(* Logix 5000 project; controller GP1 vendor 1 type 14 code 155 rev 32.11; software revision 32.01 *)
// GP1

TASK MainTask (continuous, watchdog 500 ms) : MainProgram

MODULES
   Local : vendor 1 type 14 code 155 (PointIO 0, rev 32.11)
      GP1_INPUT_MODULE_4 : 1734-IB8 (PointIO 4, rev 3.1, Input RPI 20 ms)
           Local:4:I.Data.1   // IC TOPE
           Local:4:I.Data.0   // FC TOPE
           Local:4:I.Data.3   // CAPACITIVO IZQUIERDO
           Local:4:I.Data.6   // CAPACITIVO DERECHO
      GP1_INPUT_MODULE_5 : 1734-IB8 (PointIO 5, rev 3.1, Input RPI 20 ms)
           Local:5:I.Data.2   // ARRANQUE
           Local:5:I.Data.3   // BOTON REARME
           Local:5:I.Data.1   // PARO
           Local:5:I.Data.0   // INDUCTIVO TOPE
      Discrete_IO : Embedded (PointIO 1, rev 32.11, Output RPI 20 ms)
           Local:1:I.Data.5   // IC CLAMP HORIZONTAL
           Local:1:I.Data.7   // IC CLAMP VERTICAL
           Local:1:I.Data.8   // IC NAVAJAS 3 R
           Local:1:I.Data.10   // IC CLAMP
           Local:1:I.Data.11   // FC CLAMP
           Local:1:I.Data.9   // FC NAVAJAS 3 R
           Local:1:I.Data.6   // FC CLAMP VERTICAL
           Local:1:I.Data.0   // FC NAVAJA 1
           Local:1:I.Data.1   // IC NAVAJA 1
           Local:1:I.Data.15   // FC TROQUEL
           Local:1:I.Data.2   // IC NAVAJAS 3 L
           Local:1:I.Data.4   // FC CLAMP HORIZONTAL
           Local:1:I.Data.3   // FC NAVAJAS 3 L
           Local:1:I.Data.14   // IC TROQUEL
           Local:1:I.Data.12   // FC CORTE SUPERIOR
           Local:1:I.Data.13   // IC CORTE SUPERIOR
           Local:1:O.Data.15   // GREEN
      GP1_OUTPUT_MODULE_3 : 1734-OB8 (PointIO 3, rev 3.1, Output RPI 20 ms)
      GP1_OUTPUT_MODULE_2 : 1734-OB8 (PointIO 2, rev 3.1, Output RPI 20 ms)
           Local:2:O.Data.0   // YELLOW
           Local:2:O.Data.1   // RED
           Local:2:O.Data.2   // AZUL
END_MODULES

VAR_GLOBAL   (* controller tags *)
   ACT0_OFF : BOOL := 1;   // NAVAJAS 3 R OFF
   ACT0_ON : BOOL;   // NAVAJAS 3 R ON
   ACT1_OFF : BOOL := 1;   // TROQUEL OFF
   ACT1_ON : BOOL;   // TROQUEL ON
   ACT2_OFF : BOOL := 1;   // CORTE SUPERIOR OFF
   ACT2_ON : BOOL;   // CORTE SUPERIOR ON
   ACT3_OFF : BOOL := 1;   // NAVAJA 1 OFF
   ACT3_ON : BOOL;   // NAVAJA 1 ON
   ACT4_OFF : BOOL;   // CLAMP VERTICAL OFF
   ACT4_ON : BOOL;   // CLAMP VERTICAL ON
   ACT5_OFF : BOOL := 1;   // CLAMP OFF
   ACT5_ON : BOOL;   // CLAMP ON
   ACT6_OFF : BOOL;   // CLAMP HORIZONTAL OFF
   ACT6_ON : BOOL;   // CLAMP HORIZONTAL ON
   ACT7_OFF : BOOL := 1;   // NAVAJA 3 L OFF
   ACT7_ON : BOOL;   // NAVAJA 3 L ON
   ACT8_OFF : BOOL;   // TOPE OFF
   ACT8_ON : BOOL := 1;   // TOPE ON
   AIR_ALARM : BOOL;
   ALARM_TIM : TIMER := (PRE := 5000);
   ALARMED : BOOL := 1;
   ARRANQUE_AUTO : BOOL;
   AUTO : BOOL;
   C1 : COUNTER := (ACC := 14, CU := 1, DN := 1);
   CAPACITIVE_SENSOR_1 : BOOL;
   CAPACITIVE_SENSOR_2 : BOOL;
   CND1 : BOOL;
   CND10 : BOOL;
   CND2 : BOOL;
   CND3 : BOOL;
   CND4 : BOOL;
   CND5 : BOOL;
   CND6 : BOOL;
   CND7 : BOOL;
   CND8 : BOOL;
   CND9 : BOOL;
   CORTE_VALVULA : BOOL := 1;
   CORTINA_SEG : BOOL;
   CT : COUNTER := (ACC := 9999);
   CURRENT_SCREEN : DINT;
   E_STOP : BOOL := 1;
   E_STOP_ALARM : BOOL := 1;
   EstadoHMI : DINT := 3;
   EVBI0_AUTO_OFF : BOOL;   // NAVAJAS 3 OFF AUTO
   EVBI0_AUTO_ON : BOOL;   // NAVAJAS 3 ON AUTO
   EVBI0_MAN_OFF : BOOL;   // NAVAJAS 3 OFF MANUAL
   EVBI0_MAN_ON : BOOL;   // NAVAJAS 3 ON MANUAL
   EVBI0_OFF : BOOL;   // NAVAJAS 3 OFF
   EVBI0_ON : BOOL;   // NAVAJAS 3 ON
   EVBI1_AUTO_OFF : BOOL;   // TROQUEL OFF AUTO
   EVBI1_AUTO_ON : BOOL;   // TROQUEL ON AUTO
   EVBI1_MAN_OFF : BOOL;   // TROQUEL OFF MANUAL
   EVBI1_MAN_ON : BOOL;   // TROQUEL ON MANUAL
   EVBI1_OFF : BOOL;   // TROQUEL OFF
   EVBI1_ON : BOOL;   // TROQUEL ON
   EVBI2_AUTO_OFF : BOOL;   // CLAMP OFF AUTO
   EVBI2_AUTO_ON : BOOL;   // CLAMP ON AUTO
   EVBI2_MAN_OFF : BOOL;   // CLAMP OFF MANUAL
   EVBI2_MAN_ON : BOOL;   // CLAMP ON MANUAL
   EVBI2_OFF : BOOL;   // CLAMP OFF
   EVBI2_ON : BOOL;   // CLAMP ON
   EVBI3_AUTO_OFF : BOOL;   // NAVAJA 1 OFF AUTO
   EVBI3_AUTO_ON : BOOL;   // NAVAJA 1 ON AUTO
   EVBI3_MAN_OFF : BOOL;   // NAVAJA 1 OFF MANUAL
   EVBI3_MAN_ON : BOOL;   // NAVAJA 1 ON MANUAL
   EVBI3_OFF : BOOL;   // NAVAJA 1 OFF
   EVBI3_ON : BOOL;   // NAVAJA 1 ON
   EVBI4_AUTO_OFF : BOOL;   // CLAMP VERTICAL OFF AUTO
   EVBI4_AUTO_ON : BOOL;   // CLAMP VERTICAL ON AUTO
   EVBI4_MAN_OFF : BOOL;   // CLAMP VERTICAL OFF MANUAL
   EVBI4_MAN_ON : BOOL;   // CLAMP VERTICAL ON MANUAL
   EVBI4_OFF : BOOL;   // CLAMP VERTICAL OFF
   EVBI4_ON : BOOL;   // CLAMP VERTICAL ON
   EVBI5_AUTO_OFF : BOOL;   // CORTE SUPERIOR OFF AUTO
   EVBI5_AUTO_ON : BOOL;   // CORTE SUPERIOR ON AUTO
   EVBI5_MAN_OFF : BOOL;   // CORTE SUPERIOR OFF MANUAL
   EVBI5_MAN_ON : BOOL;   // CORTE SUPERIOR ON MANUAL
   EVBI5_OFF : BOOL;   // CORTE SUPERIOR OFF
   EVBI5_ON : BOOL;   // CORTE SUPERIOR ON
   EVBI6_AUTO_OFF : BOOL;   // CLAMP HORIZONTAL OFF AUTO
   EVBI6_AUTO_ON : BOOL;   // CLAMP HORIZONTAL ON AUTO
   EVBI6_MAN_OFF : BOOL;   // CLAMP HORIZONTAL OFF MANUAL
   EVBI6_MAN_ON : BOOL;   // CLAMP HORIZONTAL ON MANUAL
   EVBI6_OFF : BOOL;   // CLAMP HORIZONTAL OFF
   EVBI6_ON : BOOL;   // CLAMP HORIZONTAL ON
   EVMONO1_AUTO_OFF : BOOL;
   EVMONO1_AUTO_ON : BOOL;   // TOPE_AUTO_ON
   EVMONO1_MAN_OFF : BOOL;
   EVMONO1_MAN_ON : BOOL;
   EVMONO_OFF : BOOL;
   EVMONO_ON : BOOL;   // TOPE ON
   EXCEDDED_TIME_FOR_CILINDERS : BOOL;
   EXCEDDED_TIME_FOR_INIT_COND : BOOL;
   FAIL_COUNT : COUNTER;
   GREEN_LIGHT : BOOL;
   INITIAL_CONDITIONS_NOT_READY : BOOL := 1;
   INITIAL_CONDITIONS_READY : BOOL;
   L_S_OK : BOOL;   // SENSOR IZQUIERDO
   LAMP : BOOL;
   LATCH_TEST : BOOL;
   LIGHT_CURTAIN : BOOL;
   MAN_SCREENS : BOOL;   // PANTALLAS MANUALES
   MANUAL : BOOL := 1;
   MSJ_CND_INIT : DINT := 8;
   NO_AIR : BOOL;
   NO_ALARM : BOOL;
   NOT_CORRECTLY_PLACED : BOOL;
   OBESTOP : BOOL;
   OK : BOOL;
   ONS1 : BOOL;
   PARO : BOOL := 1;
   Paso1 : BOOL;
   Paso10 : BOOL;
   Paso11 : BOOL;
   Paso12 : BOOL;
   Paso13 : BOOL;
   Paso14 : BOOL;
   Paso15 : BOOL;
   Paso16 : BOOL;
   Paso17 : BOOL;
   Paso18 : BOOL;
   Paso2 : BOOL;
   Paso3 : BOOL;
   Paso4 : BOOL;
   Paso5 : BOOL;
   Paso6 : BOOL;
   Paso7 : BOOL;
   Paso8 : BOOL;
   Paso9 : BOOL;
   Paso_Sec : DINT;
   PIECE_PLACED : BOOL;
   PRESOSTATO : BOOL;
   R_S_OK : BOOL;   // SENSOR DERECHO
   REARME_OK : BOOL;
   REARMY_BUTTON : BOOL;
   REARMY_TIME : TIMER := (PRE := 5);
   REARMY_WARNING : BOOL := 1;   // LUZ DE ARME
   RED_LIGHT : BOOL := 1;
   REPEATED_ALARM : BOOL;
   RESET_COUNTER : BOOL;
   RESET_LATCH_TEST : BOOL;
   SAFETY_CURTAIN : BOOL;
   SAFETY_CURTAIN_ALARM : BOOL;
   SBESTOP : BOOL;
   SENSOR1 : BOOL;
   SENSOR_TOPE : BOOL;   // TOPE DE PIEZA
   Sequence_ON : BOOL;
   Start_Sequence : BOOL;
   T1 : TIMER := (PRE := 250);
   T10 : TIMER := (PRE := 250);
   T11 : TIMER := (PRE := 250);
   T12 : TIMER := (PRE := 250);
   T13 : TIMER := (PRE := 250);
   T14 : TIMER := (PRE := 1000);
   T15 : TIMER := (PRE := 1000);
   T16 : TIMER := (PRE := 1000);
   T17 : TIMER := (PRE := 1000);
   T18 : TIMER := (PRE := 1000);
   T2 : TIMER := (PRE := 250);
   T3 : TIMER := (PRE := 250);
   T4 : TIMER := (PRE := 250);
   T5 : TIMER := (PRE := 250);
   T6 : TIMER := (PRE := 250);
   T7 : TIMER := (PRE := 250);
   T8 : TIMER := (PRE := 250);
   T9 : TIMER := (PRE := 250);
   TCLAMP : TIMER := (PRE := 250);
   TEST : BOOL;
   TEST_2 : BOOL;
   TEST_3 : BOOL;
   TEST_RESET : BOOL;
   TEST_STOP : BOOL;
   TIMOFF : TIMER := (PRE := 500);
   TIMON : TIMER := (PRE := 500);
   TIMSACC : DINT;
   TIMW1 : TIMER := (PRE := 2000);
   TIMW2 : TIMER := (PRE := 1);
   USER : DINT;
   WAITING : BOOL;
   WORKING : BOOL;
   YELLOW_LIGHT : BOOL := 1;
END_VAR

PROGRAM MainProgram   (* main routine MainRoutine *)
VAR
   BYPASS_DER : BOOL;
   BYPASS_IZQ : BOOL;
   BYPASS_TOPE : BOOL;
   BypassStatus : DINT;
   CERRARSESION : BOOL;
   ING_ACCESS : BOOL;
   LOGOUT : BOOL;
   MTTO_ACCESS : BOOL;
   RESET_COUNTERT : BOOL;
   TEMP1 : BOOL;
   TEMP2 : BOOL;
   TEMP3 : BOOL;
   USERstring : STRING;
END_VAR

ROUTINE ALARMS   (* ladder *)
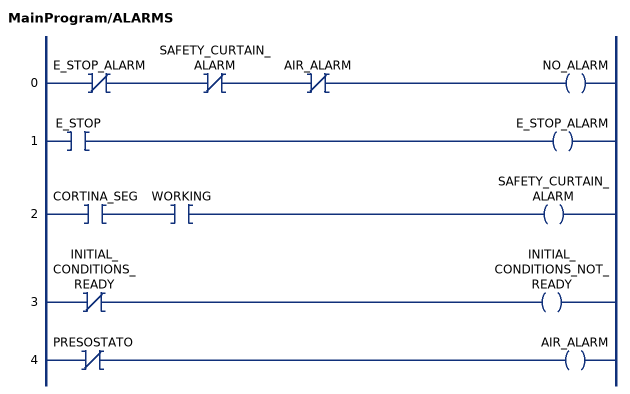
   0: XIO(E_STOP_ALARM)XIO(SAFETY_CURTAIN_ALARM)XIO(AIR_ALARM)OTE(NO_ALARM);
   1: XIC(E_STOP)OTE(E_STOP_ALARM);
   2: XIC(CORTINA_SEG)XIC(WORKING)OTE(SAFETY_CURTAIN_ALARM);
   3: XIO(INITIAL_CONDITIONS_READY)OTE(INITIAL_CONDITIONS_NOT_READY);
   4: XIO(PRESOSTATO)OTE(AIR_ALARM);
END_ROUTINE

ROUTINE AUTO_SEQUENCE   (* ladder *)
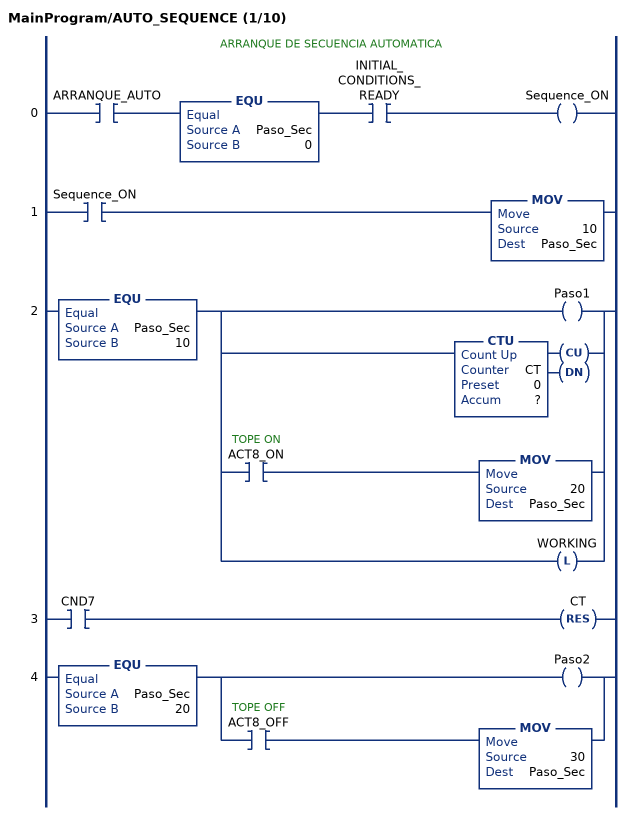
   // ARRANQUE DE SECUENCIA AUTOMATICA
   0: XIC(ARRANQUE_AUTO)EQU(Paso_Sec,0)XIC(INITIAL_CONDITIONS_READY)OTE(Sequence_ON);
   1: XIC(Sequence_ON)MOV(10,Paso_Sec);
   2: EQU(Paso_Sec,10)[OTE(Paso1) ,CTU(CT,?,?) ,XIC(ACT8_ON) MOV(20,Paso_Sec) ,OTL(WORKING) ];
   3: XIC(CND7)RES(CT);
   4: EQU(Paso_Sec,20)[OTE(Paso2) ,XIC(ACT8_OFF) MOV(30,Paso_Sec) ];
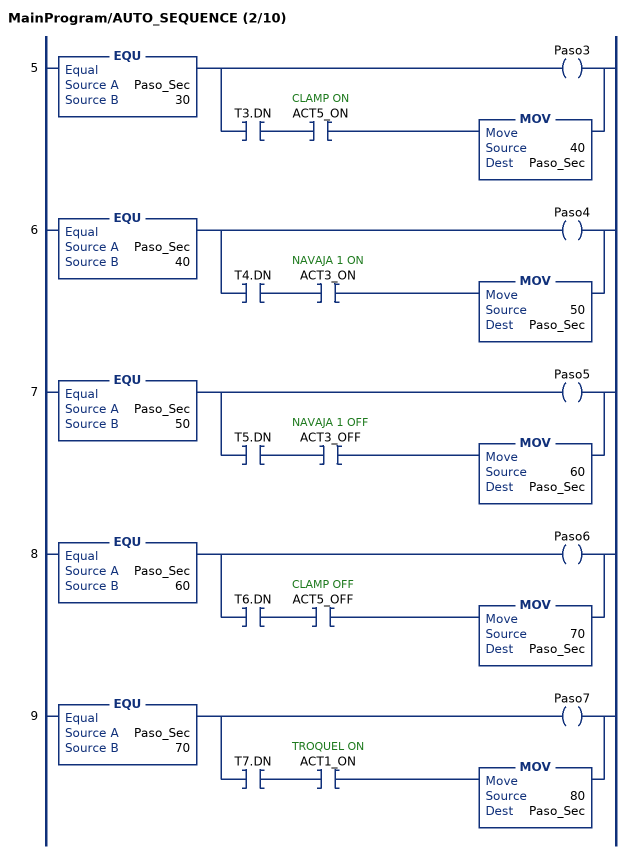
   5: EQU(Paso_Sec,30)[OTE(Paso3) ,XIC(T3.DN) XIC(ACT5_ON) MOV(40,Paso_Sec) ];
   6: EQU(Paso_Sec,40)[OTE(Paso4) ,XIC(T4.DN) XIC(ACT3_ON) MOV(50,Paso_Sec) ];
   7: EQU(Paso_Sec,50)[OTE(Paso5) ,XIC(T5.DN) XIC(ACT3_OFF) MOV(60,Paso_Sec) ];
   8: EQU(Paso_Sec,60)[OTE(Paso6) ,XIC(T6.DN) XIC(ACT5_OFF) MOV(70,Paso_Sec) ];
   9: EQU(Paso_Sec,70)[OTE(Paso7) ,XIC(T7.DN) XIC(ACT1_ON) MOV(80,Paso_Sec) ];
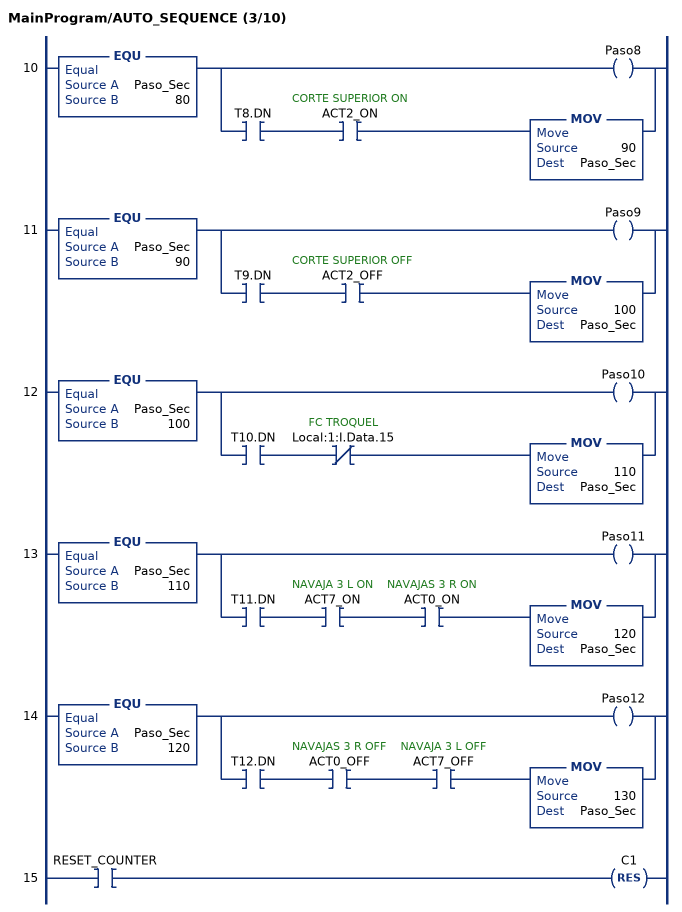
   10: EQU(Paso_Sec,80)[OTE(Paso8) ,XIC(T8.DN) XIC(ACT2_ON) MOV(90,Paso_Sec) ];
   11: EQU(Paso_Sec,90)[OTE(Paso9) ,XIC(T9.DN) XIC(ACT2_OFF) MOV(100,Paso_Sec) ];
   12: EQU(Paso_Sec,100)[OTE(Paso10) ,XIC(T10.DN) XIO(Local:1:I.Data.15) MOV(110,Paso_Sec) ];
   13: EQU(Paso_Sec,110)[OTE(Paso11) ,XIC(T11.DN) XIC(ACT7_ON) XIC(ACT0_ON) MOV(120,Paso_Sec) ];
   14: EQU(Paso_Sec,120)[OTE(Paso12) ,XIC(T12.DN) XIC(ACT0_OFF) XIC(ACT7_OFF) MOV(130,Paso_Sec) ];
   15: XIC(RESET_COUNTER)RES(C1);
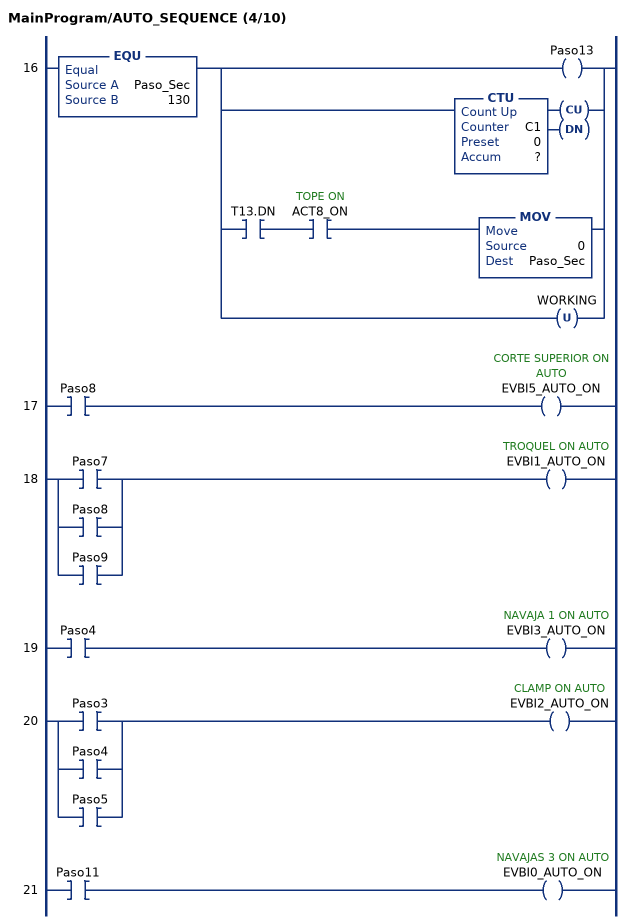
   16: EQU(Paso_Sec,130)[OTE(Paso13) ,CTU(C1,?,?) ,XIC(T13.DN) XIC(ACT8_ON) MOV(0,Paso_Sec) ,OTU(WORKING) ];
   17: XIC(Paso8)OTE(EVBI5_AUTO_ON);
   18: [XIC(Paso7) ,XIC(Paso8) ,XIC(Paso9) ]OTE(EVBI1_AUTO_ON);
   19: XIC(Paso4)OTE(EVBI3_AUTO_ON);
   20: [XIC(Paso3) ,XIC(Paso4) ,XIC(Paso5) ]OTE(EVBI2_AUTO_ON);
   21: XIC(Paso11)OTE(EVBI0_AUTO_ON);
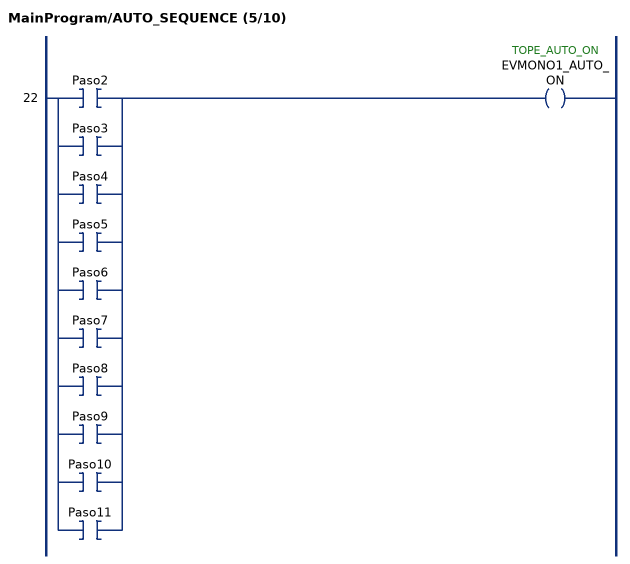
   22: [XIC(Paso2) ,XIC(Paso3) ,XIC(Paso4) ,XIC(Paso5) ,XIC(Paso6) ,XIC(Paso7) ,XIC(Paso8) ,XIC(Paso9) ,XIC(Paso10) ,XIC(Paso11) ]OTE(EVMONO1_AUTO_ON);
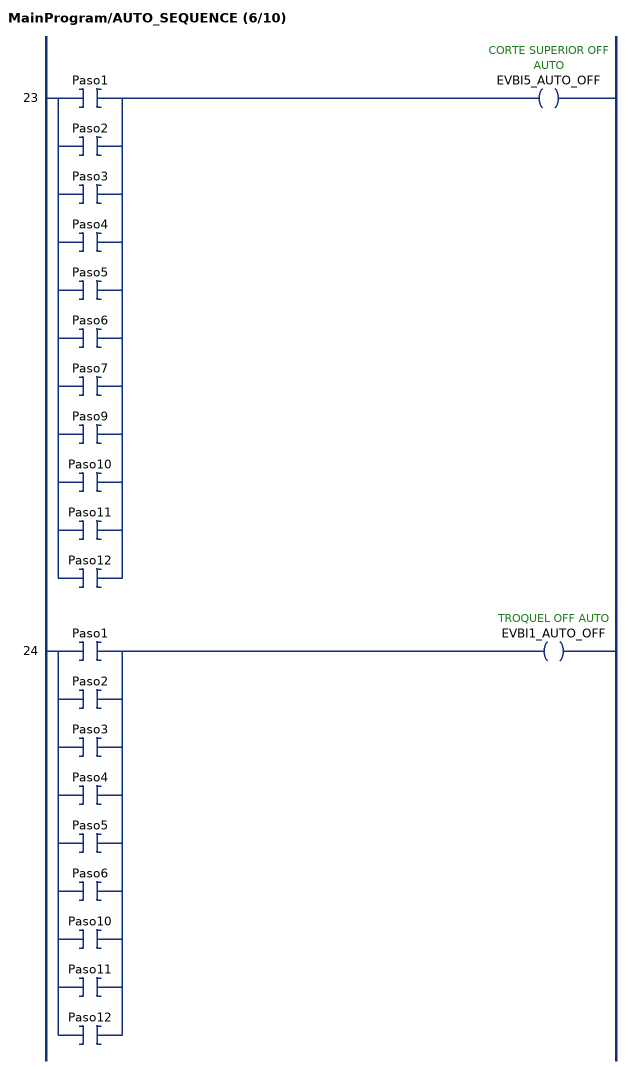
   23: [XIC(Paso1) ,XIC(Paso2) ,XIC(Paso3) ,XIC(Paso4) ,XIC(Paso5) ,XIC(Paso6) ,XIC(Paso7) ,XIC(Paso9) ,XIC(Paso10) ,XIC(Paso11) ,XIC(Paso12) ]OTE(EVBI5_AUTO_OFF);
   24: [XIC(Paso1) ,XIC(Paso2) ,XIC(Paso3) ,XIC(Paso4) ,XIC(Paso5) ,XIC(Paso6) ,XIC(Paso10) ,XIC(Paso11) ,XIC(Paso12) ]OTE(EVBI1_AUTO_OFF);
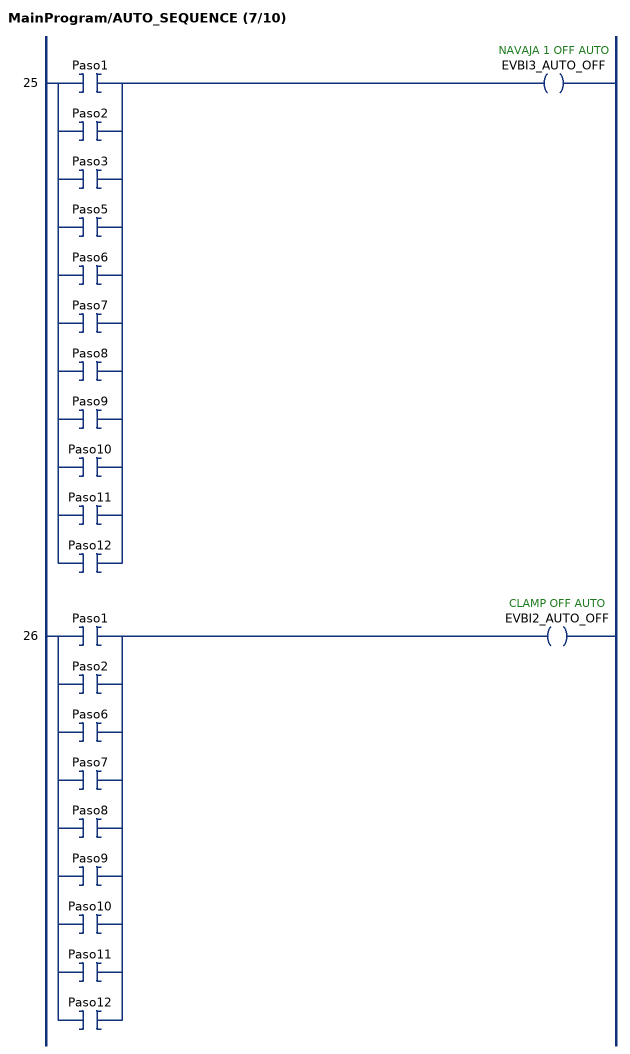
   25: [XIC(Paso1) ,XIC(Paso2) ,XIC(Paso3) ,XIC(Paso5) ,XIC(Paso6) ,XIC(Paso7) ,XIC(Paso8) ,XIC(Paso9) ,XIC(Paso10) ,XIC(Paso11) ,XIC(Paso12) ]OTE(EVBI3_AUTO_OFF);
   26: [XIC(Paso1) ,XIC(Paso2) ,XIC(Paso6) ,XIC(Paso7) ,XIC(Paso8) ,XIC(Paso9) ,XIC(Paso10) ,XIC(Paso11) ,XIC(Paso12) ]OTE(EVBI2_AUTO_OFF);
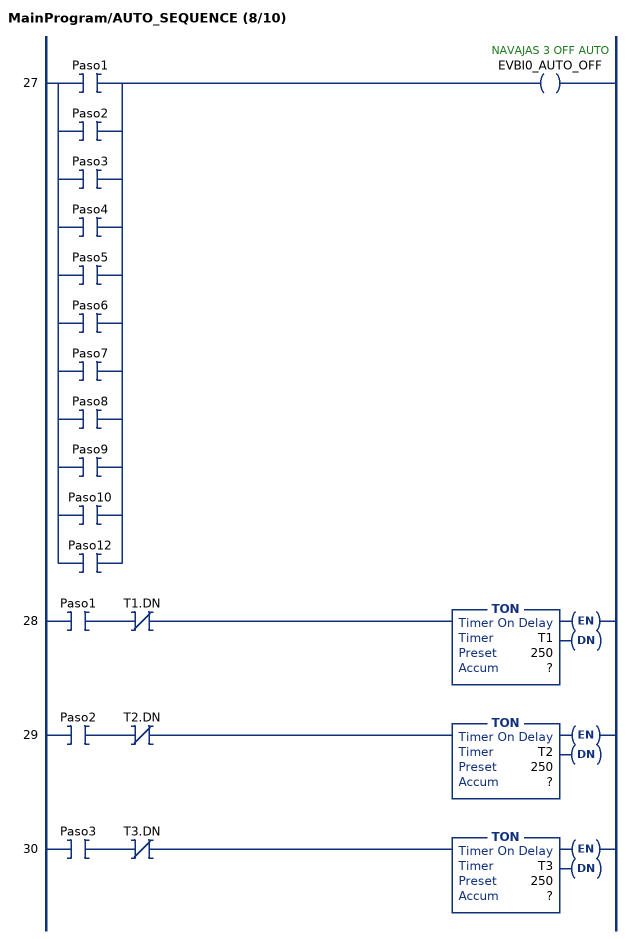
   27: [XIC(Paso1) ,XIC(Paso2) ,XIC(Paso3) ,XIC(Paso4) ,XIC(Paso5) ,XIC(Paso6) ,XIC(Paso7) ,XIC(Paso8) ,XIC(Paso9) ,XIC(Paso10) ,XIC(Paso12) ]OTE(EVBI0_AUTO_OFF);
   28: XIC(Paso1)XIO(T1.DN)TON(T1,?,?);
   29: XIC(Paso2)XIO(T2.DN)TON(T2,?,?);
   30: XIC(Paso3)XIO(T3.DN)TON(T3,?,?);
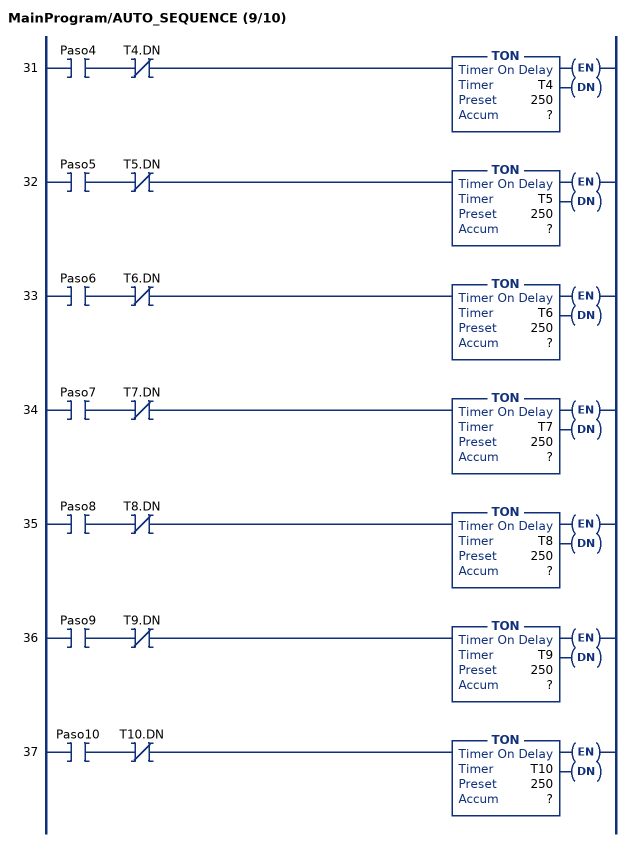
   31: XIC(Paso4)XIO(T4.DN)TON(T4,?,?);
   32: XIC(Paso5)XIO(T5.DN)TON(T5,?,?);
   33: XIC(Paso6)XIO(T6.DN)TON(T6,?,?);
   34: XIC(Paso7)XIO(T7.DN)TON(T7,?,?);
   35: XIC(Paso8)XIO(T8.DN)TON(T8,?,?);
   36: XIC(Paso9)XIO(T9.DN)TON(T9,?,?);
   37: XIC(Paso10)XIO(T10.DN)TON(T10,?,?);
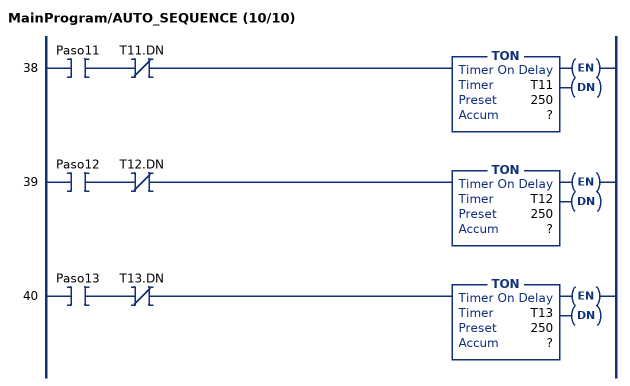
   38: XIC(Paso11)XIO(T11.DN)TON(T11,?,?);
   39: XIC(Paso12)XIO(T12.DN)TON(T12,?,?);
   40: XIC(Paso13)XIO(T13.DN)TON(T13,?,?);
END_ROUTINE

ROUTINE INPUTS   (* ladder *)
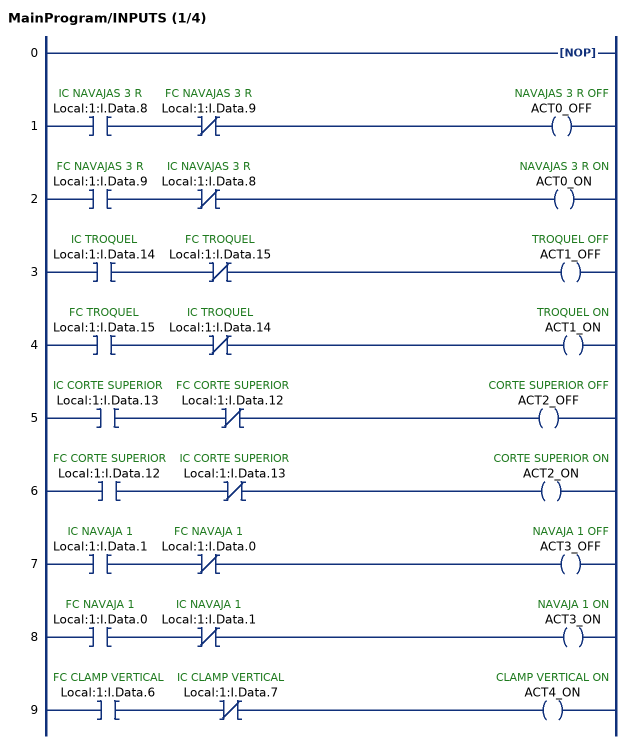
   0: NOP();
   1: XIC(Local:1:I.Data.8)XIO(Local:1:I.Data.9)OTE(ACT0_OFF);
   2: XIC(Local:1:I.Data.9)XIO(Local:1:I.Data.8)OTE(ACT0_ON);
   3: XIC(Local:1:I.Data.14)XIO(Local:1:I.Data.15)OTE(ACT1_OFF);
   4: XIC(Local:1:I.Data.15)XIO(Local:1:I.Data.14)OTE(ACT1_ON);
   5: XIC(Local:1:I.Data.13)XIO(Local:1:I.Data.12)OTE(ACT2_OFF);
   6: XIC(Local:1:I.Data.12)XIO(Local:1:I.Data.13)OTE(ACT2_ON);
   7: XIC(Local:1:I.Data.1)XIO(Local:1:I.Data.0)OTE(ACT3_OFF);
   8: XIC(Local:1:I.Data.0)XIO(Local:1:I.Data.1)OTE(ACT3_ON);
   9: XIC(Local:1:I.Data.6)XIO(Local:1:I.Data.7)OTE(ACT4_ON);
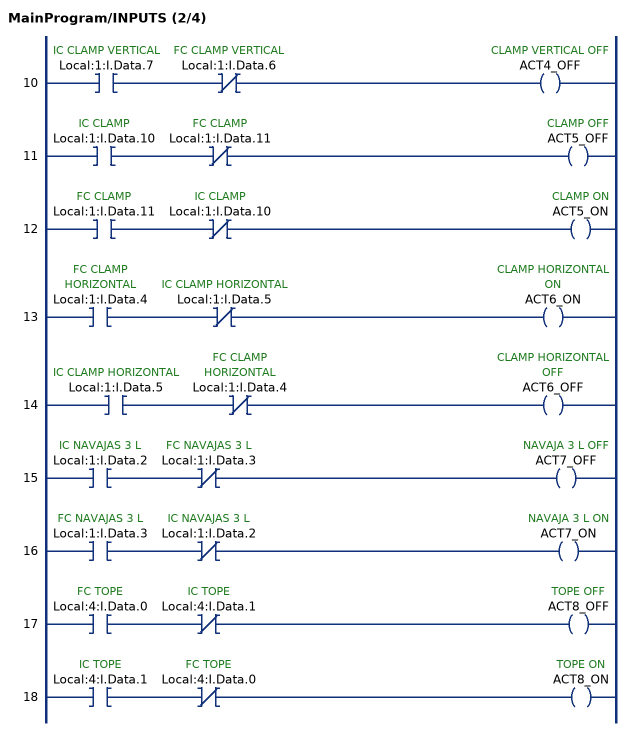
   10: XIC(Local:1:I.Data.7)XIO(Local:1:I.Data.6)OTE(ACT4_OFF);
   11: XIC(Local:1:I.Data.10)XIO(Local:1:I.Data.11)OTE(ACT5_OFF);
   12: XIC(Local:1:I.Data.11)XIO(Local:1:I.Data.10)OTE(ACT5_ON);
   13: XIC(Local:1:I.Data.4)XIO(Local:1:I.Data.5)OTE(ACT6_ON);
   14: XIC(Local:1:I.Data.5)XIO(Local:1:I.Data.4)OTE(ACT6_OFF);
   15: XIC(Local:1:I.Data.2)XIO(Local:1:I.Data.3)OTE(ACT7_OFF);
   16: XIC(Local:1:I.Data.3)XIO(Local:1:I.Data.2)OTE(ACT7_ON);
   17: XIC(Local:4:I.Data.0)XIO(Local:4:I.Data.1)OTE(ACT8_OFF);
   18: XIC(Local:4:I.Data.1)XIO(Local:4:I.Data.0)OTE(ACT8_ON);
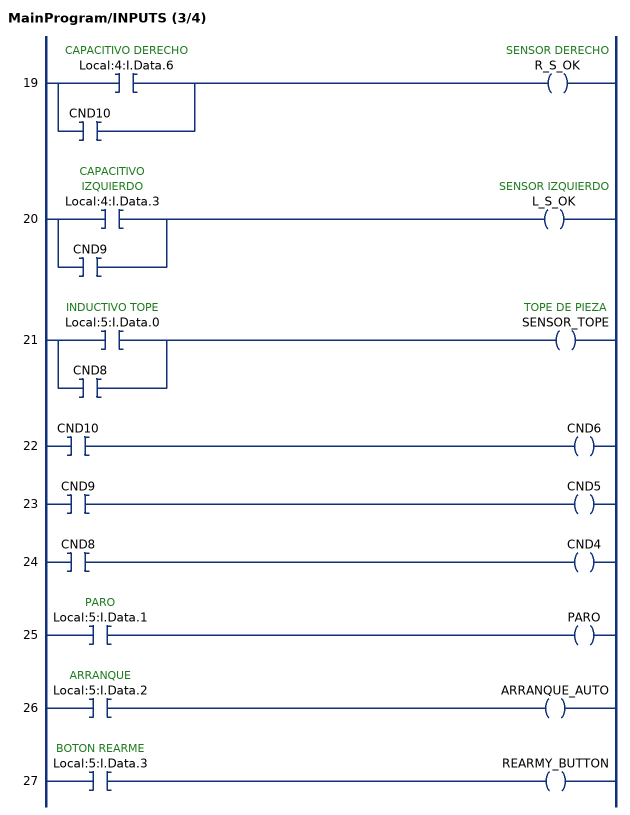
   19: [XIC(Local:4:I.Data.6) ,XIC(CND10) ]OTE(R_S_OK);
   20: [XIC(Local:4:I.Data.3) ,XIC(CND9) ]OTE(L_S_OK);
   21: [XIC(Local:5:I.Data.0) ,XIC(CND8) ]OTE(SENSOR_TOPE);
   22: XIC(CND10)OTE(CND6);
   23: XIC(CND9)OTE(CND5);
   24: XIC(CND8)OTE(CND4);
   25: XIC(Local:5:I.Data.1)OTE(PARO);
   26: XIC(Local:5:I.Data.2)OTE(ARRANQUE_AUTO);
   27: XIC(Local:5:I.Data.3)OTE(REARMY_BUTTON);
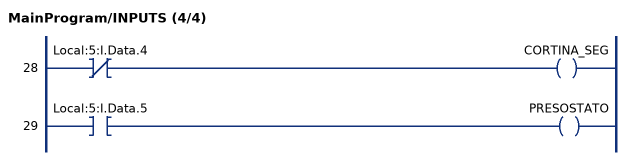
   28: XIO(Local:5:I.Data.4)OTE(CORTINA_SEG);
   29: XIC(Local:5:I.Data.5)OTE(PRESOSTATO);
END_ROUTINE

ROUTINE MACHINE_STATES   (* ladder *)
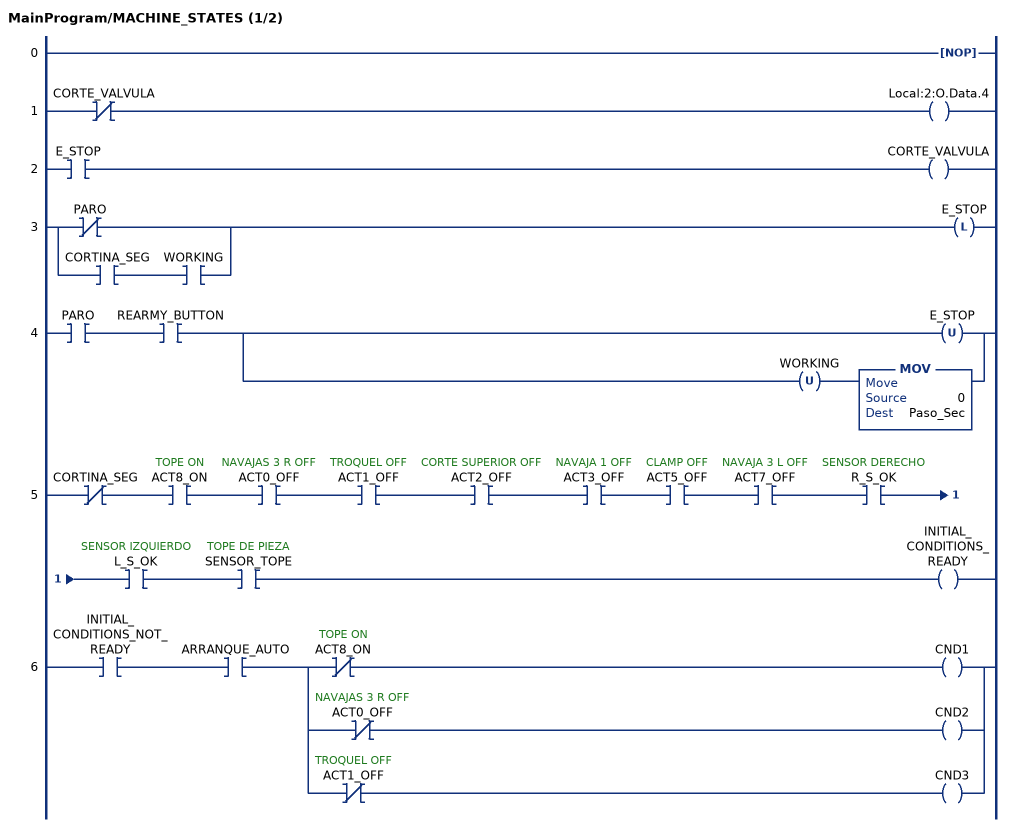
   0: NOP();
   1: XIO(CORTE_VALVULA)OTE(Local:2:O.Data.4);
   2: XIC(E_STOP)OTE(CORTE_VALVULA);
   3: [XIO(PARO) ,XIC(CORTINA_SEG) XIC(WORKING) ]OTL(E_STOP);
   4: XIC(PARO)XIC(REARMY_BUTTON)[OTU(E_STOP) ,OTU(WORKING) MOV(0,Paso_Sec) ];
   5: XIO(CORTINA_SEG)XIC(ACT8_ON)XIC(ACT0_OFF)XIC(ACT1_OFF)XIC(ACT2_OFF)XIC(ACT3_OFF)XIC(ACT5_OFF)XIC(ACT7_OFF)XIC(R_S_OK)XIC(L_S_OK)XIC(SENSOR_TOPE)OTE(INITIAL_CONDITIONS_READY);
   6: XIC(INITIAL_CONDITIONS_NOT_READY)XIC(ARRANQUE_AUTO)[XIO(ACT8_ON) OTE(CND1) ,XIO(ACT0_OFF) OTE(CND2) ,XIO(ACT1_OFF) OTE(CND3) ];
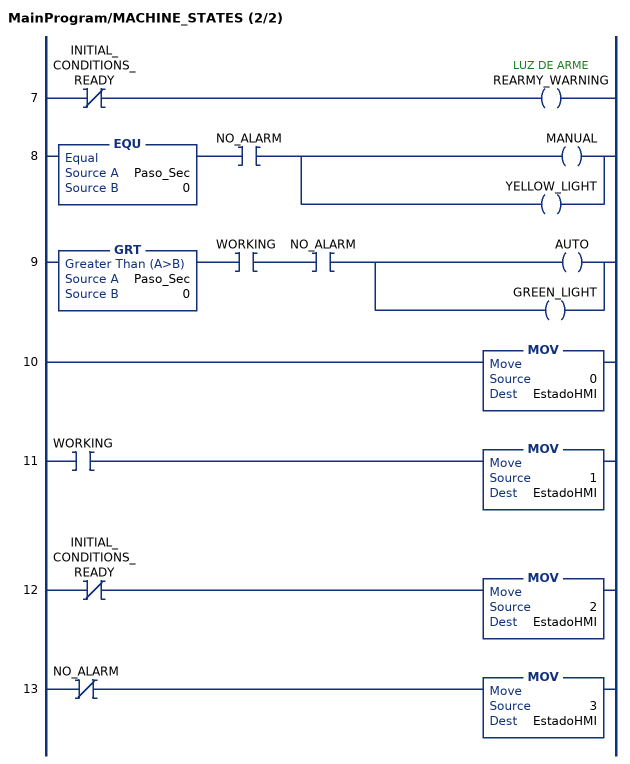
   7: XIO(INITIAL_CONDITIONS_READY)OTE(REARMY_WARNING);
   8: EQU(Paso_Sec,0)XIC(NO_ALARM)[OTE(MANUAL) ,OTE(YELLOW_LIGHT) ];
   9: GRT(Paso_Sec,0)XIC(WORKING)XIC(NO_ALARM)[OTE(AUTO) ,OTE(GREEN_LIGHT) ];
   10: MOV(0,EstadoHMI);
   11: XIC(WORKING)MOV(1,EstadoHMI);
   12: XIO(INITIAL_CONDITIONS_READY)MOV(2,EstadoHMI);
   13: XIO(NO_ALARM)MOV(3,EstadoHMI);
END_ROUTINE

ROUTINE MainRoutine   (* ladder *)
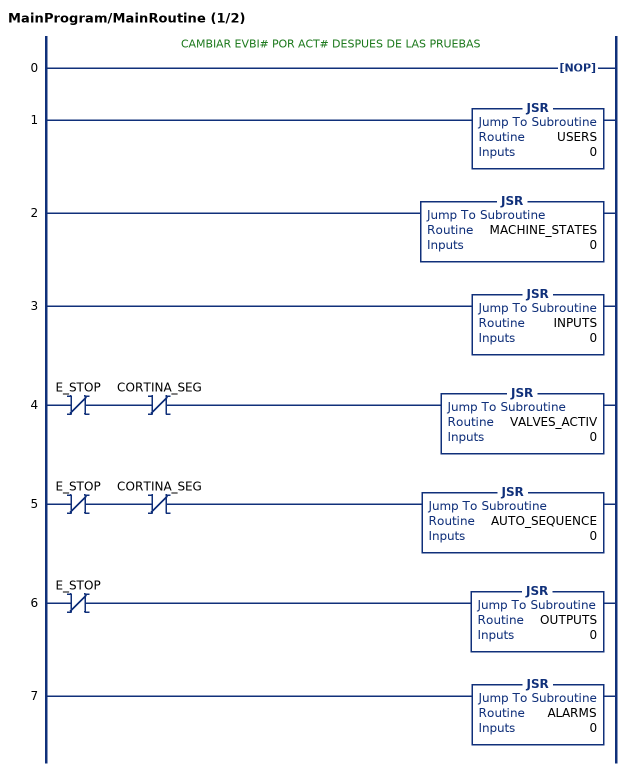
   // CAMBIAR EVBI# POR ACT# DESPUES DE LAS PRUEBAS
   0: NOP();
   1: JSR(USERS,0);
   2: JSR(MACHINE_STATES,0);
   3: JSR(INPUTS,0);
   4: XIO(E_STOP)XIO(CORTINA_SEG)JSR(VALVES_ACTIV,0);
   5: XIO(E_STOP)XIO(CORTINA_SEG)JSR(AUTO_SEQUENCE,0);
   6: XIO(E_STOP)JSR(OUTPUTS,0);
   7: JSR(ALARMS,0);
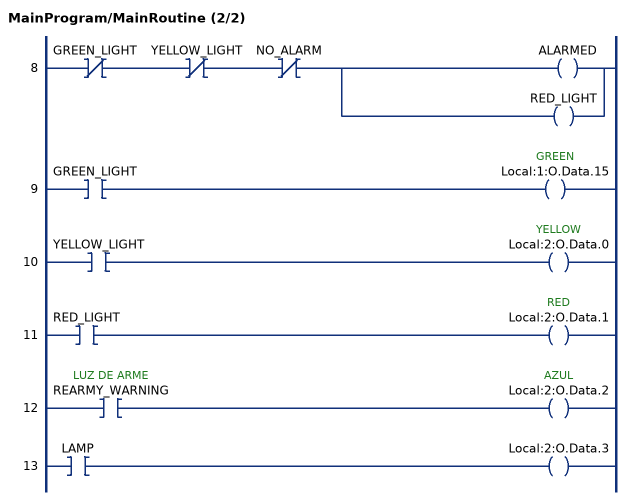
   8: XIO(GREEN_LIGHT)XIO(YELLOW_LIGHT)XIO(NO_ALARM)[OTE(ALARMED) ,OTE(RED_LIGHT) ];
   9: XIC(GREEN_LIGHT)OTE(Local:1:O.Data.15);
   10: XIC(YELLOW_LIGHT)OTE(Local:2:O.Data.0);
   11: XIC(RED_LIGHT)OTE(Local:2:O.Data.1);
   12: XIC(REARMY_WARNING)OTE(Local:2:O.Data.2);
   13: XIC(LAMP)OTE(Local:2:O.Data.3);
END_ROUTINE
